FUNCTION_BLOCK TEvent_DayChanged EXTENDS TEventBase IMPLEMENTS IEvent
VAR
	Now: TIMESTRUCT;
    Handler : IEventHandler_OnDayChanged;
END_VAR

METHOD  CallHandler
VAR_INPUT
    HandlerBase : IEventHandlerBase;
END_VAR
IF __QUERYINTERFACE(HandlerBase,Handler) THEN
    Handler.OnDayChanged(Now);
END_IF
END_METHOD

METHOD  IsHandlerSupported : BOOL
VAR_INPUT
    EventHandler : IEventHandlerBase;
END_VAR
IF __QUERYINTERFACE(EventHandler,Handler) THEN
    IsHandlerSupported := TRUE;
END_IF
END_METHOD

METHOD RaiseEx
VAR_INPUT
	Now: TIMESTRUCT;
END_VAR
THIS^.Now := Now;
SUPER^.Raise();
END_METHOD

END_FUNCTION_BLOCK

(* stored: Version 1.1.0.1, ProductVersion 3.1.4024.3
   POU TEvent_DayChanged: Id {b9788094-e17d-0058-0b1f-d0e90b67c34f}, SpecialFunc None
   Method CallHandler: Id {0b6c4cb4-cb40-0423-2a05-fdf1eab7426f}
   Method IsHandlerSupported: Id {ac0dad3b-4e7d-0604-2f1c-135f9ecb5506}
   Method RaiseEx: Id {aedee585-cfd0-0333-1f86-c0ca8e9aa6ba} *)
